PROGRAM INTERNAL MAIN
VAR
END_VAR

END_PROGRAM

(* stored: Version 1.1.0.1
   POU MAIN: Id {3a2fb5d7-16dd-05a6-2ac8-813c36e4ace1}, SpecialFunc None *)
